// TIA Portal V19 export
TYPE "AreaConfig"
// stored: Access Published
   STRUCT
      TimeOutStopImmediate { ExternalAccessible := 'False'; ExternalVisible := 'False'; ExternalWritable := 'False'} : Time := t#1500ms;   // Timeout for receive ack stop in phase from machines when a stop immediate is required
      TimeOutStopInPhase { ExternalAccessible := 'False'; ExternalVisible := 'False'; ExternalWritable := 'False'} : Time := T#10S;   // Timeout for receive ack stop in phase from machines when a normal stop is required
      TimeOutStopProgrammed { ExternalAccessible := 'False'; ExternalVisible := 'False'; ExternalWritable := 'False'} : Time := T#300s;   // Timeout for receive ack stop programmed from machines
      TimeOutResetAlarms { ExternalAccessible := 'False'; ExternalVisible := 'False'; ExternalWritable := 'False'} : Time := T#1s;   // Time of reset alarms to machine
   END_STRUCT;
END_TYPE
